(* PLC project  *)

CONFIGURATION StepIM_A
END_CONFIGURATION
